{attribute 'GeneratedUsingTerminal: EL2521-0000-1016'}
{attribute addProperty BoxType "EL2521-0000-1016"}
{attribute addProperty Id "Set_counterAT %Q*BOOL1Set_counter_valueAT %Q*UINT2"}
{attribute addProperty CRC "610056523"}
{attribute addProperty Size "3"}
TYPE ENC_Control_compact_245CB94B :
STRUCT
	{attribute addProperty Name "Set_counter"}
	Set_counter AT %Q* : BOOL;
	{attribute addProperty Name "Set_counter_value"}
	Set_counter_value AT %Q* : UINT;
END_STRUCT
END_TYPE

(* stored: Version 1.2.0.0, ProductVersion 3.1.4024.9
   DUT ENC_Control_compact_245CB94B: Id {883ade21-5b14-4f35-91f1-6f3f3278cc74} *)
